// TIA Portal V16 export
// export: Created 2023-01-03T15:35:07.7910522Z, ExportSetting WithDefaults, DisplayName Totally Integrated Automation Portal, DisplayVersion V16, DisplayName TIA Portal Version Control Interface, DisplayVersion V16, DisplayName TIA Portal Openness, DisplayVersion V16, DisplayName STEP 7 Professional, DisplayVersion V16, DisplayName STEP 7 Safety, DisplayVersion V16, DisplayName WinCC Advanced, DisplayVersion V16
FUNCTION "MOTOR_SPEEDCONTROL" : Void   // FC4, LAD
{ S7_Optimized_Access := 'TRUE' }
VERSION : 0.1
// stored: AutoNumber true, IsIECCheckEnabled false, SetENOAutomatically false, UDAEnableTagReadback false
   VAR_INPUT
      Speed_SP_rpm : Real;
   END_VAR
   VAR_OUTPUT
      Output : Int;
      Return_Value : Bool;
   END_VAR
   VAR_TEMP
      Speed_sp_in_range : Bool;
      Normalized : Real;
   END_VAR
BEGIN

REGION Network 1
   // FIRST CHECK THAT THE SPEED INPUT IS WITHIN THE RANGE OR NOT. IF NOT THEN SEND '0' TO THE OUTPUT.
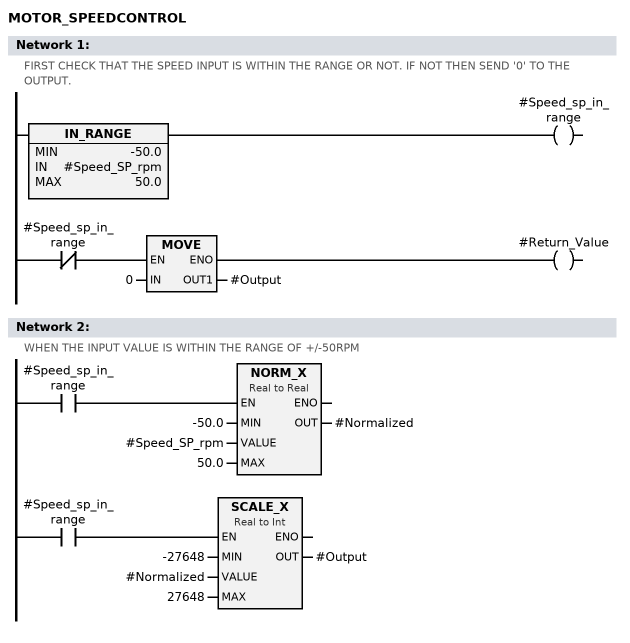
   RUNG wire#powerrail
      { S7_Templates := "SrcType := Real" } InRange(min := -50.0, in := #Speed_SP_rpm, max := 50.0)
      Coil( #Speed_sp_in_range )
   END_RUNG
   RUNG wire#powerrail
      I_Contact( #Speed_sp_in_range )
      Move(in := 0, out1 => #Output)
      Coil( #Return_Value )
   END_RUNG
   // the same network as SCL:
   #Speed_sp_in_range := (-50.0 <= #Speed_SP_rpm) AND (#Speed_SP_rpm <= 50.0);
   IF NOT #Speed_sp_in_range THEN #Output := 0; END_IF;
   #Return_Value := NOT #Speed_sp_in_range;
END_REGION

REGION Network 2
   // WHEN THE INPUT VALUE IS WITHIN THE RANGE OF +/-50RPM
   RUNG wire#powerrail
      Contact( #Speed_sp_in_range )
      { S7_Templates := "[SrcType := Real, DestType := Real]" } Normalize(min := -50.0, value := #Speed_SP_rpm, max := 50.0, out => #Normalized)
   END_RUNG
   RUNG wire#powerrail
      Contact( #Speed_sp_in_range )
      { S7_Templates := "[SrcType := Real, DestType := Int]" } Scale(min := -27648, value := #Normalized, max := 27648, out => #Output)
   END_RUNG
   // the same network as SCL:
   IF #Speed_sp_in_range THEN
       #Normalized := NORM_X(MIN := -50.0, VALUE := #Speed_SP_rpm, MAX := 50.0);
       #Output := SCALE_X(MIN := -27648, VALUE := #Normalized, MAX := 27648);
   END_IF;
END_REGION
END_FUNCTION
